{attribute 'linkalways'} 
{attribute 'no_explicit_call' := 'This FB is a CLASS and must be accessed using methods or properties'}
{attribute 'enable_dynamic_creation'}
FUNCTION_BLOCK _ETcVnHoughMethod EXTENDS EnumDatatypeBase
VAR
	localData : ETcVnHoughMethod;
	activeData : REFERENCE TO ETcVnHoughMethod;
	enumBaseDatatype : _DINT(localData);
END_VAR

METHOD PRIVATE AddLocalEnumeration
VAR_INPUT
	Enumeration : T_MAXSTRING;
	Value : ETcVnHoughMethod;
END_VAR
AddEnumeration(Enumeration, Value);
END_METHOD

PROPERTY PUBLIC Address : PVOID
GET
Address := ADR(activeData);
END_GET
END_PROPERTY

METHOD PUBLIC ClearReference
VAR_INPUT
END_VAR
activeData REF= localData;
SetBaseDatatypeReference();
END_METHOD

METHOD PUBLIC Clone : I_Datatype
VAR
    pClone : POINTER TO _ETcVnHoughMethod;
END_VAR
pClone := __NEW(_ETcVnHoughMethod(InitialValue := Value));
Clone := pClone^;
END_METHOD

METHOD FB_init : BOOL
VAR_INPUT
	bInitRetains : BOOL; // if TRUE, the retain variables are initialized (warm start / cold start)
	bInCopyCode : BOOL;  // if TRUE, the instance afterwards gets moved into the copy code (online change)
	InitialValue : ETcVnHoughMethod;
END_VAR
localData := InitialValue;
AddBaseDatatype(enumBaseDatatype);
ClearReference();

AddLocalEnumeration('TCVN_HM_STANDARD', ETcVnHoughMethod.TCVN_HM_STANDARD);
AddLocalEnumeration('TCVN_HM_PROBABILISTIC', ETcVnHoughMethod.TCVN_HM_PROBABILISTIC);
AddLocalEnumeration('TCVN_HM_MULTI_SCALE', ETcVnHoughMethod.TCVN_HM_MULTI_SCALE);
AddLocalEnumeration('TCVN_HM_GRADIENT', ETcVnHoughMethod.TCVN_HM_GRADIENT);
AddLocalEnumeration('TCVN_HM_GRADIENT_ALT', ETcVnHoughMethod.TCVN_HM_GRADIENT_ALT);
END_METHOD

PROPERTY PUBLIC Identifier : T_MAXSTRING
GET
Identifier := 'ETcVnHoughMethod';
END_GET
END_PROPERTY

METHOD IsEnumeratorValueEqual : BOOL
VAR_INPUT
	Enumerator : I_KeyValueForwardEnumerator;
END_VAR
VAR
	storedValue : ETcVnHoughMethod;
END_VAR
IF NOT Enumerator.TryGet(storedValue) THEN
	RETURN;
END_IF

IsEnumeratorValueEqual := storedValue = activeData;
END_METHOD

METHOD PUBLIC MakeReferenceTo
VAR_INPUT
	ReferenceTarget : REFERENCE TO ETcVnHoughMethod;
END_VAR
activeData REF= ReferenceTarget;
SetBaseDatatypeReference();
END_METHOD

METHOD PROTECTED SetBaseDatatypeReference
VAR_INPUT
END_VAR
enumBaseDatatype.MakeReferenceTo(activeData);
END_METHOD

PROPERTY PUBLIC Size : UDINT
GET
Size := SIZEOF(activeData);
END_GET
END_PROPERTY

METHOD TryMakeReferenceTo : BOOL
VAR_INPUT
	Target : I_Datatype;
END_VAR
VAR
	targetAsEnum : I_EnumDatatype;
	pTargetData : POINTER TO ETcVnHoughMethod;
END_VAR
IF NOT Target.TryResolveAsEnumDatatype(targetAsEnum) THEN
	RETURN;
END_IF

IF targetAsEnum.Identifier <> Identifier THEN
	RETURN;
END_IF

pTargetData := Target.Address;
activeData REF= pTargetData^;
SetBaseDatatypeReference();
TryMakeReferenceTo := TRUE;
END_METHOD

PROPERTY PUBLIC Value : ETcVnHoughMethod
GET
Value := activeData;
END_GET
SET
activeData := Value;
END_SET
END_PROPERTY

END_FUNCTION_BLOCK

(* stored: Version 1.1.0.1
   POU _ETcVnHoughMethod: Id {358dba64-1ebe-4605-8b8e-2586668c4fac}, SpecialFunc None
   Folder Constructor: Id {39590a9d-1683-4275-95b8-6ad8dd275893}
   Folder Private: Id {9678c1a1-ca04-4592-a92e-0dc3bfcbf81b}
   Folder Protected: Id {207ab40d-f5d2-4d05-b776-3d0d68c21a30}
   Method AddLocalEnumeration: Id {6e97ca05-3746-4939-b4fa-66287aa7df70}
   Property Address: Id {80f41edf-d9d9-406e-955a-6c99539a2d2f}
   Get Get: Id {7f6a9249-2fd8-43c2-b4e3-e2269dd86930}
   Method ClearReference: Id {77748971-9658-44a4-8f39-00b4a6afa288}
   Method Clone: Id {22bafe7c-20ee-480f-b996-ec43935f0a38}
   Method FB_init: Id {3ebbfa96-35c2-4789-85d9-0274e955711c}
   Property Identifier: Id {5469aefb-87e6-49f3-b458-2efd971023c3}
   Get Get: Id {f2968c5b-bf61-4dd7-abbe-a8be42d421ac}
   Method IsEnumeratorValueEqual: Id {b4fbe8e3-6129-4f78-aca3-d40f04078f77}
   Method MakeReferenceTo: Id {dae7ce23-1806-427d-897e-144a80ecde37}
   Method SetBaseDatatypeReference: Id {ff65cd0b-5d15-4e78-92ee-da7f628901a1}
   Property Size: Id {117e28dd-7292-406f-bf76-2a783c113843}
   Get Get: Id {c59d5775-e36f-44b1-87f6-4594c33761cb}
   Method TryMakeReferenceTo: Id {b3825500-3720-4c60-80cb-3ee21ade7fe0}
   Property Value: Id {f6001d12-1834-4cf9-ad02-cce8f0458efc}
   Get Get: Id {8c68df21-5869-4101-b351-91baeb2b5033}
   Set Set: Id {4b830454-c302-45f9-893f-b059ae2bf4b4} *)
